// TIA Portal V16 export
// export: Created 2021-08-16T20:43:06.6006589Z, ExportSetting WithDefaults, DisplayName Totally Integrated Automation Portal, DisplayVersion V16, DisplayName TIA Portal Version Control Interface, DisplayVersion V16, DisplayName TIA Portal Openness, DisplayVersion V16, DisplayName STEP 7 Professional, DisplayVersion V16, DisplayName STEP 7 Safety, DisplayVersion V16, DisplayName WinCC Advanced, DisplayVersion V16
VAR_GLOBAL   // PLC tag table "Default tag table"
   STOP AT %M0.0 : Bool;
   START AT %M0.1 : Bool;
   "READY 2 Run" AT %M0.2 : Bool;
   "Actual pcs" AT %MW2 : Int;
   "Another Piece" AT %M0.3 : Bool;
   "Full Box" AT %M0.4 : Bool;
   PulseFlag AT %M0.5 : Bool;
   PulseOut AT %M0.6 : Bool;
   "Box Capacity" AT %MW8 : Int;
   "Sensor Final" AT %M1.2 : Bool;
   "Sensor Middle" AT %M1.1 : Bool;
   "Sensor Start" AT %M1.0 : Bool;
   "Pcs in Extrusion" AT %MW4 : Int;
   "Extrusions in Box" AT %MW6 : Int;
   "Actual extrusion" AT %MW10 : Int;
   "Coveyor 2 Delay" AT %MD12 : Time;
END_VAR
VAR_GLOBAL CONSTANT   // user constants
   "Krabica mala" : Int := 150;
   "Krabica velka" : Int := 250;
END_VAR
